Omron CX-Programmer project NewProject (CX-Programmer 9.10)

# PLC IO_Test: CJ2M CPU32
I/O table (CPU CJ2M-CPU32): rack 0 slot 11 CJ2M-EIP21

## Program NewProgram1 (cyclic task 0)
Local symbols
be1 2.00 BOOL
be10 2.09 BOOL
be11 2.10 BOOL
be12 2.11 BOOL
be13 2.12 BOOL
be14 2.13 BOOL
be15 2.14 BOOL
be16 2.15 BOOL
be2 2.01 BOOL
be3 2.02 BOOL
be4 2.03 BOOL
be5 2.04 BOOL
be6 2.05 BOOL
be7 2.06 BOOL
be8 2.07 BOOL
be9 2.08 BOOL
ki1 3.00 BOOL
ki10 3.09 BOOL
ki11 3.10 BOOL
ki12 3.11 BOOL
ki13 3.12 BOOL
ki14 3.13 BOOL
ki15 3.14 BOOL
ki16 3.15 BOOL
ki2 3.01 BOOL
ki3 3.02 BOOL
ki4 3.03 BOOL
ki5 3.04 BOOL
ki6 3.05 BOOL
ki7 3.06 BOOL
ki8 3.07 BOOL
ki9 3.08 BOOL

### Section Section1

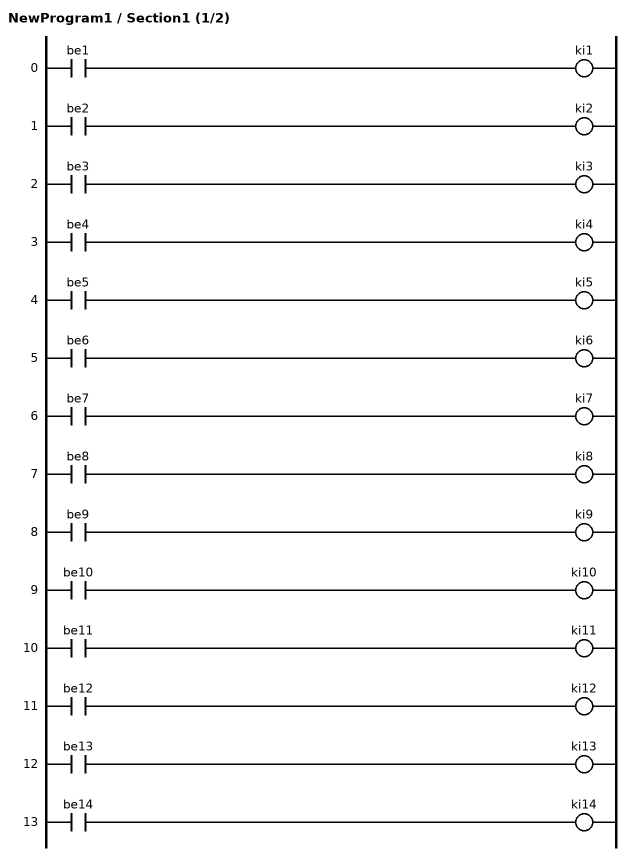
; rung 0
LD be1
OUT ki1
; rung 1
LD be2
OUT ki2
; rung 2
LD be3
OUT ki3
; rung 3
LD be4
OUT ki4
; rung 4
LD be5
OUT ki5
; rung 5
LD be6
OUT ki6
; rung 6
LD be7
OUT ki7
; rung 7
LD be8
OUT ki8
; rung 8
LD be9
OUT ki9
; rung 9
LD be10
OUT ki10
; rung 10
LD be11
OUT ki11
; rung 11
LD be12
OUT ki12
; rung 12
LD be13
OUT ki13
; rung 13
LD be14
OUT ki14

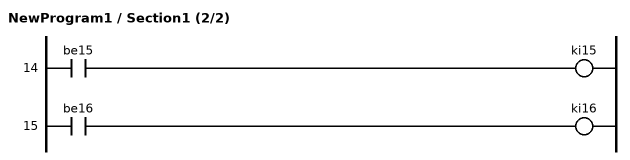
; rung 14
LD be15
OUT ki15
; rung 15
LD be16
OUT ki16

### Section END
; rung 0
END(001)